// TIA Portal V17 export
// export: Created 2022-04-06T07:28:38.6030972Z, ExportSetting WithDefaults, DisplayName Totally Integrated Automation Portal, DisplayVersion V17, DisplayName TIA Portal Openness, DisplayVersion V17, DisplayName TIA Portal Version Control Interface, DisplayVersion V17, DisplayName TIA Portal Test Suite Advanced, DisplayVersion V17, DisplayName SINAMICS Startdrive Advanced, DisplayVersion V17, DisplayName SINAMICS Startdrive G130, G150, S120, S150, SINAMICS MV, S210, DisplayVersion V17, DisplayName SINAMICS Startdrive G110M, G120, G120C, G120D, G120P, G115D, DisplayVersion V17, DisplayName STEP 7 Professional, DisplayVersion V17, DisplayName STEP 7 Safety, DisplayVersion V17, DisplayName WinCC Advanced / Unified PC, DisplayVersion V17
FUNCTION_BLOCK "SINA_FFB1"   // FB6, F_FBD
{ S7_Optimized_Access := 'TRUE' }
VERSION : 0.1
// stored: AutoNumber true, IsIECCheckEnabled true, UDAEnableTagReadback false
   VAR_INPUT
      tel30Status : "LDrvSafe_typeSinaSTlg30Status";
      acknowledge : Bool;
      releaseEstop : Bool := true;
      releaseGate : Bool := true;
      enableMode : Bool := true;
   END_VAR
   VAR_OUTPUT
      tel30Control : "LDrvSafe_typeSinaSTlg30Control";
   END_VAR
   VAR
      statSlsTof : TOF;
      statTrue : Bool;
      statSto : Bool;
      statSs1 : Bool;
      statSs2 : Bool;
      statSos : Bool;
      statSls : Bool;
      statSlp : Bool;
      statSLA : Bool;
      statProfiSafeStatus : "LDrvSafe_typeSinaSTlg30Control";
   END_VAR
BEGIN

REGION Network 1
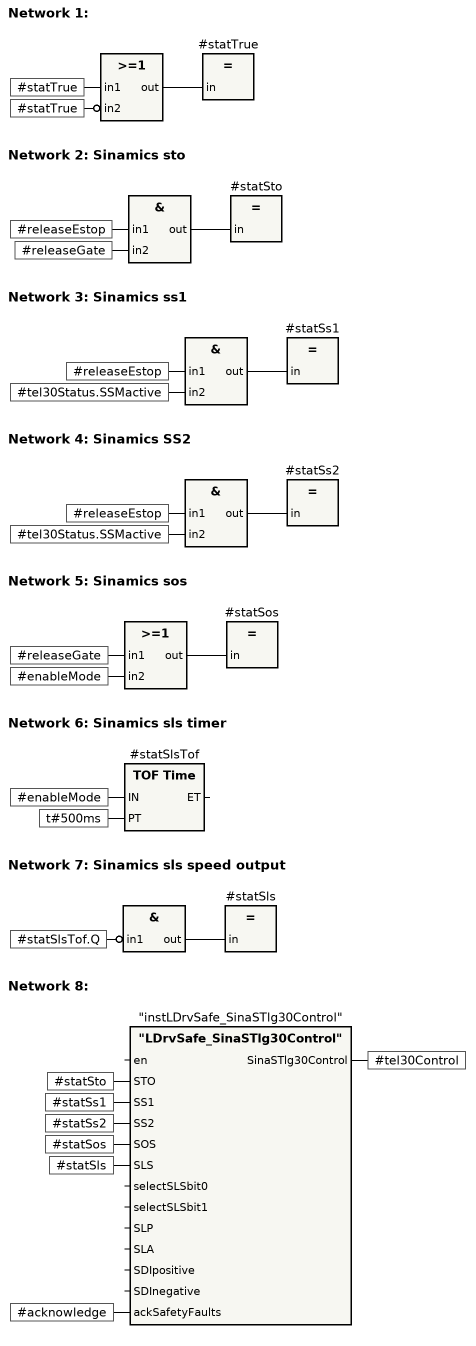
   #statTrue := #statTrue OR NOT #statTrue;
END_REGION

REGION Network 2: Sinamics sto
   #statSto := #releaseEstop AND #releaseGate;
END_REGION

REGION Network 3: Sinamics ss1
   #statSs1 := #releaseEstop AND #tel30Status.SSMactive;
END_REGION

REGION Network 4: Sinamics SS2
   #statSs2 := #releaseEstop AND #tel30Status.SSMactive;
END_REGION

REGION Network 5: Sinamics sos
   #statSos := #releaseGate OR #enableMode;
END_REGION

REGION Network 6: Sinamics sls timer
   #statSlsTof.TOF(IN := #enableMode, PT := t#500ms);
END_REGION

REGION Network 7: Sinamics sls speed output
   #statSls := NOT #statSlsTof.Q;
END_REGION

REGION Network 8
   "instLDrvSafe_SinaSTlg30Control"(STO := #statSto,   // "LDrvSafe_SinaSTlg30Control"
                           SS1 := #statSs1,
                           SS2 := #statSs2,
                           SOS := #statSos,
                           SLS := #statSls,
                           ackSafetyFaults := #acknowledge,
                           SinaSTlg30Control => #tel30Control);
END_REGION
END_FUNCTION_BLOCK
